TYPE ST_PlateOrder :
STRUCT
	PlateOrder:INT;
	BoxStatus:E_BoxStatus;
END_STRUCT
END_TYPE

(* stored: Version 1.1.0.1, ProductVersion 3.1.4024.13
   DUT ST_PlateOrder: Id {6d6ddf2e-6309-45cf-8c4f-e8b0a2bed4ee} *)
